Universal Robots PolyScope program: comb_run.urp

Program comb_run (installation=default directory=/programs/usbdisk createdIn=5.12.4.1101661 lastSavedIn=5.12.4.1101661)
Robot Program (runOnlyOnce=true)
  Script file /programs/usbdisk/comb.script
    | def draw_svg():
    |   draw_z = 0.074940
    |   # home
    |   movel(p[0.598550, -0.129200, 0.105150, 2.249000, -2.194000, 0.000000], a=0.8, v=0.25, r=0.0)
    |   # stroke 0 (form id 0): simpleline
    |   movel(p[0.756629, -0.217706, 0.118080, 2.230000, -2.212000, 0.000000], a=0.8, v=0.25, r=0.0)
    |   movep(p[0.756629, -0.217706, draw_z, 2.230000, -2.212000, 0.000000], a=0.5, v=0.02, r=0.015000)
    |   movep(p[0.756169, -0.016748, draw_z, 2.230000, -2.212000, 0.000000], a=0.5, v=0.02, r=0.000000)
    |   movel(p[0.756169, -0.016748, 0.118080, 2.230000, -2.212000, 0.000000], a=0.8, v=0.25, r=0.0)
    |   # stroke 1 (form id 1): simpleline
    |   movel(p[0.736591, -0.218031, 0.118080, 2.230000, -2.212000, 0.000000], a=0.8, v=0.25, r=0.0)
    |   movep(p[0.736591, -0.218031, draw_z, 2.230000, -2.212000, 0.000000], a=0.5, v=0.02, r=0.015000)
    |   movep(p[0.736131, -0.017074, draw_z, 2.230000, -2.212000, 0.000000], a=0.5, v=0.02, r=0.000000)
    |   movel(p[0.736131, -0.017074, 0.118080, 2.230000, -2.212000, 0.000000], a=0.8, v=0.25, r=0.0)
    |   # stroke 2 (form id 2): simpleline
    |   movel(p[0.716553, -0.218357, 0.118080, 2.230000, -2.212000, 0.000000], a=0.8, v=0.25, r=0.0)
    |   movep(p[0.716553, -0.218357, draw_z, 2.230000, -2.212000, 0.000000], a=0.5, v=0.02, r=0.015000)
    |   movep(p[0.716092, -0.017400, draw_z, 2.230000, -2.212000, 0.000000], a=0.5, v=0.02, r=0.000000)
    |   movel(p[0.716092, -0.017400, 0.118080, 2.230000, -2.212000, 0.000000], a=0.8, v=0.25, r=0.0)
    |   # stroke 3 (form id 3): simpleline
    |   movel(p[0.696515, -0.218683, 0.118080, 2.230000, -2.212000, 0.000000], a=0.8, v=0.25, r=0.0)
    |   movep(p[0.696515, -0.218683, draw_z, 2.230000, -2.212000, 0.000000], a=0.5, v=0.02, r=0.015000)
    |   movep(p[0.696054, -0.017726, draw_z, 2.230000, -2.212000, 0.000000], a=0.5, v=0.02, r=0.000000)
    |   movel(p[0.696054, -0.017726, 0.118080, 2.230000, -2.212000, 0.000000], a=0.8, v=0.25, r=0.0)
    |   # stroke 4 (form id 4): simpleline
    |   movel(p[0.669338, -0.219125, 0.118080, 2.230000, -2.212000, 0.000000], a=0.8, v=0.25, r=0.0)
    |   movep(p[0.669338, -0.219125, draw_z, 2.230000, -2.212000, 0.000000], a=0.5, v=0.02, r=0.015000)
    |   movep(p[0.668878, -0.018168, draw_z, 2.230000, -2.212000, 0.000000], a=0.5, v=0.02, r=0.000000)
    |   movel(p[0.668878, -0.018168, 0.118080, 2.230000, -2.212000, 0.000000], a=0.8, v=0.25, r=0.0)
    |   # stroke 5 (form id 5): simpleline
    |   movel(p[0.654310, -0.219370, 0.118080, 2.230000, -2.212000, 0.000000], a=0.8, v=0.25, r=0.0)
    |   movep(p[0.654310, -0.219370, draw_z, 2.230000, -2.212000, 0.000000], a=0.5, v=0.02, r=0.015000)
    |   movep(p[0.653849, -0.018413, draw_z, 2.230000, -2.212000, 0.000000], a=0.5, v=0.02, r=0.000000)
    |   movel(p[0.653849, -0.018413, 0.118080, 2.230000, -2.212000, 0.000000], a=0.8, v=0.25, r=0.0)
    |   # stroke 6 (form id 6): simpleline
    |   movel(p[0.639281, -0.219614, 0.118080, 2.230000, -2.212000, 0.000000], a=0.8, v=0.25, r=0.0)
    |   movep(p[0.639281, -0.219614, draw_z, 2.230000, -2.212000, 0.000000], a=0.5, v=0.02, r=0.015000)
    |   movep(p[0.638821, -0.018657, draw_z, 2.230000, -2.212000, 0.000000], a=0.5, v=0.02, r=0.000000)
    |   movel(p[0.638821, -0.018657, 0.118080, 2.230000, -2.212000, 0.000000], a=0.8, v=0.25, r=0.0)
    |   # stroke 7 (form id 7): simpleline
    |   movel(p[0.624253, -0.219859, 0.118080, 2.230000, -2.212000, 0.000000], a=0.8, v=0.25, r=0.0)
    |   movep(p[0.624253, -0.219859, draw_z, 2.230000, -2.212000, 0.000000], a=0.5, v=0.02, r=0.015000)
    |   movep(p[0.623792, -0.018902, draw_z, 2.230000, -2.212000, 0.000000], a=0.5, v=0.02, r=0.000000)
    |   movel(p[0.623792, -0.018902, 0.118080, 2.230000, -2.212000, 0.000000], a=0.8, v=0.25, r=0.0)
    |   # stroke 8 (form id 8): simpleline
    |   movel(p[0.597076, -0.220301, 0.118080, 2.230000, -2.212000, 0.000000], a=0.8, v=0.25, r=0.0)
    |   movep(p[0.597076, -0.220301, draw_z, 2.230000, -2.212000, 0.000000], a=0.5, v=0.02, r=0.015000)
    |   movep(p[0.596615, -0.019344, draw_z, 2.230000, -2.212000, 0.000000], a=0.5, v=0.02, r=0.000000)
    |   movel(p[0.596615, -0.019344, 0.118080, 2.230000, -2.212000, 0.000000], a=0.8, v=0.25, r=0.0)
    |   # stroke 9 (form id 9): simpleline
    |   movel(p[0.585053, -0.220496, 0.118080, 2.230000, -2.212000, 0.000000], a=0.8, v=0.25, r=0.0)
    |   movep(p[0.585053, -0.220496, draw_z, 2.230000, -2.212000, 0.000000], a=0.5, v=0.02, r=0.015000)
    |   movep(p[0.584593, -0.019539, draw_z, 2.230000, -2.212000, 0.000000], a=0.5, v=0.02, r=0.000000)
    |   movel(p[0.584593, -0.019539, 0.118080, 2.230000, -2.212000, 0.000000], a=0.8, v=0.25, r=0.0)
    |   # stroke 10 (form id 10): simpleline
    |   movel(p[0.573030, -0.220692, 0.118080, 2.230000, -2.212000, 0.000000], a=0.8, v=0.25, r=0.0)
    |   movep(p[0.573030, -0.220692, draw_z, 2.230000, -2.212000, 0.000000], a=0.5, v=0.02, r=0.015000)
    |   movep(p[0.572570, -0.019735, draw_z, 2.230000, -2.212000, 0.000000], a=0.5, v=0.02, r=0.000000)
    |   movel(p[0.572570, -0.019735, 0.118080, 2.230000, -2.212000, 0.000000], a=0.8, v=0.25, r=0.0)
    |   # stroke 11 (form id 11): simpleline
    |   movel(p[0.561007, -0.220888, 0.118080, 2.230000, -2.212000, 0.000000], a=0.8, v=0.25, r=0.0)
    |   movep(p[0.561007, -0.220888, draw_z, 2.230000, -2.212000, 0.000000], a=0.5, v=0.02, r=0.015000)
    |   movep(p[0.560547, -0.019930, draw_z, 2.230000, -2.212000, 0.000000], a=0.5, v=0.02, r=0.000000)
    |   movel(p[0.560547, -0.019930, 0.118080, 2.230000, -2.212000, 0.000000], a=0.8, v=0.25, r=0.0)
    |   # stroke 12 (form id 12): simpleline
    |   movel(p[0.533831, -0.221330, 0.118080, 2.230000, -2.212000, 0.000000], a=0.8, v=0.25, r=0.0)
    |   movep(p[0.533831, -0.221330, draw_z, 2.230000, -2.212000, 0.000000], a=0.5, v=0.02, r=0.015000)
    |   movep(p[0.533370, -0.020372, draw_z, 2.230000, -2.212000, 0.000000], a=0.5, v=0.02, r=0.000000)
    |   movel(p[0.533370, -0.020372, 0.118080, 2.230000, -2.212000, 0.000000], a=0.8, v=0.25, r=0.0)
    |   # stroke 13 (form id 13): simpleline
    |   movel(p[0.523812, -0.221493, 0.118080, 2.230000, -2.212000, 0.000000], a=0.8, v=0.25, r=0.0)
    |   movep(p[0.523812, -0.221493, draw_z, 2.230000, -2.212000, 0.000000], a=0.5, v=0.02, r=0.015000)
    |   movep(p[0.523351, -0.020535, draw_z, 2.230000, -2.212000, 0.000000], a=0.5, v=0.02, r=0.000000)
    |   movel(p[0.523351, -0.020535, 0.118080, 2.230000, -2.212000, 0.000000], a=0.8, v=0.25, r=0.0)
    |   # stroke 14 (form id 14): simpleline
    |   movel(p[0.513793, -0.221656, 0.118080, 2.230000, -2.212000, 0.000000], a=0.8, v=0.25, r=0.0)
    |   movep(p[0.513793, -0.221656, draw_z, 2.230000, -2.212000, 0.000000], a=0.5, v=0.02, r=0.015000)
    |   movep(p[0.513332, -0.020698, draw_z, 2.230000, -2.212000, 0.000000], a=0.5, v=0.02, r=0.000000)
    |   movel(p[0.513332, -0.020698, 0.118080, 2.230000, -2.212000, 0.000000], a=0.8, v=0.25, r=0.0)
    |   # stroke 15 (form id 15): simpleline
    |   movel(p[0.503774, -0.221819, 0.118080, 2.230000, -2.212000, 0.000000], a=0.8, v=0.25, r=0.0)
    |   movep(p[0.503774, -0.221819, draw_z, 2.230000, -2.212000, 0.000000], a=0.5, v=0.02, r=0.015000)
    |   movep(p[0.503313, -0.020861, draw_z, 2.230000, -2.212000, 0.000000], a=0.5, v=0.02, r=0.000000)
    |   movel(p[0.503313, -0.020861, 0.118080, 2.230000, -2.212000, 0.000000], a=0.8, v=0.25, r=0.0)
    |   # stroke 16 (form id 16): simpleline
    |   movel(p[0.476597, -0.222261, 0.118080, 2.230000, -2.212000, 0.000000], a=0.8, v=0.25, r=0.0)
    |   movep(p[0.476597, -0.222261, draw_z, 2.230000, -2.212000, 0.000000], a=0.5, v=0.02, r=0.015000)
    |   movep(p[0.476137, -0.021303, draw_z, 2.230000, -2.212000, 0.000000], a=0.5, v=0.02, r=0.000000)
    |   movel(p[0.476137, -0.021303, 0.118080, 2.230000, -2.212000, 0.000000], a=0.8, v=0.25, r=0.0)
    |   # stroke 17 (form id 17): simpleline
    |   movel(p[0.468582, -0.222391, 0.118080, 2.230000, -2.212000, 0.000000], a=0.8, v=0.25, r=0.0)
    |   movep(p[0.468582, -0.222391, draw_z, 2.230000, -2.212000, 0.000000], a=0.5, v=0.02, r=0.015000)
    |   movep(p[0.468121, -0.021434, draw_z, 2.230000, -2.212000, 0.000000], a=0.5, v=0.02, r=0.000000)
    |   movel(p[0.468121, -0.021434, 0.118080, 2.230000, -2.212000, 0.000000], a=0.8, v=0.25, r=0.0)
    |   # stroke 18 (form id 18): simpleline
    |   movel(p[0.460567, -0.222521, 0.118080, 2.230000, -2.212000, 0.000000], a=0.8, v=0.25, r=0.0)
    |   movep(p[0.460567, -0.222521, draw_z, 2.230000, -2.212000, 0.000000], a=0.5, v=0.02, r=0.015000)
    |   movep(p[0.460106, -0.021564, draw_z, 2.230000, -2.212000, 0.000000], a=0.5, v=0.02, r=0.000000)
    |   movel(p[0.460106, -0.021564, 0.118080, 2.230000, -2.212000, 0.000000], a=0.8, v=0.25, r=0.0)
    |   # stroke 19 (form id 19): simpleline
    |   movel(p[0.452551, -0.222652, 0.118080, 2.230000, -2.212000, 0.000000], a=0.8, v=0.25, r=0.0)
    |   movep(p[0.452551, -0.222652, draw_z, 2.230000, -2.212000, 0.000000], a=0.5, v=0.02, r=0.015000)
    |   movep(p[0.452091, -0.021694, draw_z, 2.230000, -2.212000, 0.000000], a=0.5, v=0.02, r=0.000000)
    |   movel(p[0.452091, -0.021694, 0.118080, 2.230000, -2.212000, 0.000000], a=0.8, v=0.25, r=0.0)
    |   # park
    |   movel(p[0.598550, -0.129200, 0.105150, 2.249000, -2.194000, 0.000000], a=0.8, v=0.25, r=0.0)
    | end
    | draw_svg()
